Fanuc KAREL source: kt00167.KL

-- PROVISIONAL review KL for V940-1; original PC SHA256 b05bbcced28466c4428460e54d167bdcd94f30490629d55467ae5c3c293d1819
-- Incomplete behavior may be omitted. Consult companion uncertainty JSON. Do not deploy.
PROGRAM KT00167
%NOLOCKGROUP
VAR
  I1 : INTEGER
  OUT : INTEGER
-- UNRESOLVED_DECL H2 type=002017
BEGIN
  -- V9_ZERO_TABLE_METADATA_HINT layout=0001; no indexed target words; source/name/runtime held
  -- UNRESOLVED_PC offsets 5-16; opcodes 2E,23
  -- UNRESOLVED_PC offsets 21-35; opcodes 2E,22,9D,33,B4
  -- UNRESOLVED_PC offsets 40-62; opcodes 21,22,9D,33,B3,56,23
  -- UNRESOLVED_PC offsets 67-71; opcodes 7F
END KT00167
